(* CoDeSys 2.3.9.50 project: 7B.pr6 *)
(* Libraries: STANDARD.LB6 5.6.98 12:03:02 *)

(* POU MAIN, LD *)
PROGRAM MAIN
VAR
	Switch1 AT %IX0.0: BOOL;
	Switch2 AT %IX0.1: BOOL;
	BothOn AT %QX0.0: BOOL;
	PartPresent AT %IX0.2: BOOL;
	PartOn AT %QX0.1: BOOL;
	DrillingStarts AT %QX0.2: BOOL;
END_VAR
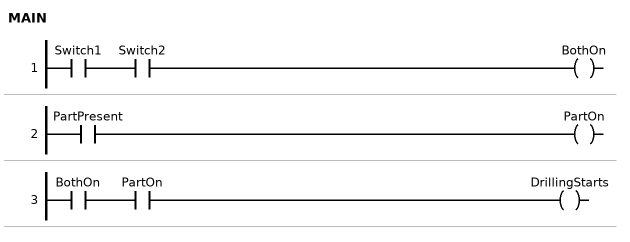
_LD_ (* Ladder Diagram *)
NETWORK 1
	[Switch1] - [Switch2] --- (BothOn)
NETWORK 2
	[PartPresent] --- (PartOn)
NETWORK 3
	[BothOn] - [PartOn] --- (DrillingStarts)
_END_LD_
(* the same logic as Structured Text *)
(* Network 1 *)
BothOn := Switch1 AND Switch2;
(* Network 2 *)
PartOn := PartPresent;
(* Network 3 *)
DrillingStarts := BothOn AND PartOn;
END_PROGRAM
